FUNCTION_BLOCK EspPacketProcessor IMPLEMENTS ITF_Cyclic
VAR
	
	Udp							: ITF_UdpConnection;
	UdpReceiveBuffer			: REFERENCE TO ARRAY [0..TCPADS_MAXUDP_BUFFSIZE - 1] OF BYTE;
	LastCheckedIndex			: UDINT;
	List						: ITF_LinkedList;
	PacketsReceived				: ULINT;
	
	ReceivedPacketType			: BYTE;
	ReceivedPacketLocation		: PVOID;
	ReceivedPacketLength		: UINT;
	
	hr1							: HRESULT;
	OpenUdpConnection			: HRESULT;
	hr3							: HRESULT;
	
	TestPacket					: EspUdpPayload1;
	CurrentEsp32				: ITF_EspHost;
	
END_VAR
VAR CONSTANT
	StartDelimiter1				: BYTE := 2;
	StartDelimiter2				: BYTE := 181;
	EndDelimiter1				: BYTE := 91;
	EndDelimiter2				: BYTE := 03;
	PacketTypePosition			: BYTE := 37;
END_VAR

METHOD PRIVATE ClearBufferAtLocation : BOOL
VAR_INPUT
	PayloadLength			: UINT;
	PayloadLocation			: PVOID;
END_VAR
VAR
	i	: UDINT;
END_VAR

IF MEMSET(PayloadLocation, 0, PayloadLength) > 0 THEN

	ClearBufferAtLocation := TRUE;
	
ELSE
	
	ClearBufferAtLocation := FALSE;
	
END_IF

RETURN;
END_METHOD

METHOD ClearEntireBuffer : BOOL
VAR_INPUT
END_VAR
VAR
	i	: UDINT;
END_VAR

FOR i := 0 TO TCPADS_MAXUDP_BUFFSIZE - 1 BY 1 DO

	UdpReceiveBuffer[i] := 0;

END_FOR
END_METHOD

METHOD PRIVATE CopyPacketIntoStructure : BOOL
VAR_INPUT
	PayloadType				: BYTE;
	PayloadLength			: UINT;
	PayloadLocation			: PVOID;
END_VAR
CASE PayloadType OF
	
	1:
	
		MEMCPY(ADR(TestPacket), PayloadLocation, PayloadLength); 
		
		TestPacket.Start := HeaderEndianSwap(TestPacket.Start);
		
		TestPacket.End := TailEndianSwap(TestPacket.End);
		
		CopyPacketIntoStructure := TRUE;
		
		
		
	2:
	
		//
	
	
	
	3:
		
		//
	
	
	
END_CASE
END_METHOD

METHOD CreateEsp : BOOL
VAR_INPUT
END_VAR
END_METHOD

METHOD CyclicUpdate : BOOL
VAR
END_VAR

Udp.CyclicUpdate();
	

IF TryOpenConnection() = S_OK AND_THEN
	TryFindPacketInBuffer(ReceivedPacketType, ReceivedPacketLength, ReceivedPacketLocation) = S_OK AND_THEN
	CopyPacketIntoStructure(ReceivedPacketType, ReceivedPacketLength, ReceivedPacketLocation) AND_THEN 
	ClearBufferAtLocation(ReceivedPacketLength, ReceivedPacketLocation) THEN
	
	
	;
	
	
END_IF






// 
// hr1 := TryFindAPacketInBuffer(ReceivedPacketType, ReceivedPacketLength, ReceivedPacketLocation);
// 
// IF hr1 = S_OK THEN
// 	
// 	IF CopyPacketIntoStructure(ReceivedPacketType, ReceivedPacketLength, ReceivedPacketLocation) THEN
// 		
// 		ClearBufferAtLocation(ReceivedPacketLength, ReceivedPacketLocation);
// 		
// 	END_IF
// 
// END_IF
END_METHOD

//FB_Init is always available implicitly and it is used primarily for initialization.
//The return value is not evaluated. For a specific influence, you can also declare the
//methods explicitly and provide additional code there with the standard initialization
//code. You can evaluate the return value.
METHOD FB_Init: BOOL
VAR_INPUT
    bInitRetains: BOOL; // TRUE: the retain variables are initialized (reset warm / reset cold)
    bInCopyCode: BOOL;  // TRUE: the instance will be copied to the copy code afterward (online change)   
	UdpSocket	: ITF_UdpConnection;
	EspList		: ITF_LinkedList;
END_VAR
Udp := UdpSocket;
UdpReceiveBuffer REF= Udp.ReceiveBufferReference;
List := EspList;
END_METHOD

METHOD IsAcceptingData : BOOL
VAR_INPUT
END_VAR
IsAcceptingData := Udp.IsConnected();

RETURN;
END_METHOD

METHOD PRIVATE MatchUidToEsp : ITF_EspHost
VAR_INPUT
	Header	: EspUdpStart;
END_VAR
VAR
	Length	: UINT;
	i		: UINT;
	Node	: ITF_Node;
	Ptr		: POINTER TO EspHost;
	Esp		: ITF_EspHost;
	Uid		: ULINT;
END_VAR

Length := List.GetListLength();

IF Length = 0 THEN
	
	MatchUidToEsp := 0;
		
	RETURN;

END_IF

FOR i := 1 TO Length BY 1 DO

	Node := List.GetNode(i);	
	
	Ptr := Node.GetMyPointer();
	
	Esp := Ptr^;
	
	IF Esp = 0 THEN
		
		MatchUidToEsp := 0;
		
		RETURN;
		
	END_IF
	
	Uid := Esp.Uid;
	
	IF Uid = Header.SlaveUid THEN // = uid in buffer 
		
		MatchUidToEsp := Esp;
		
		RETURN;
		
	END_IF

END_FOR
END_METHOD

METHOD PRIVATE TryFindPacketInBuffer : HRESULT
VAR_INPUT
	PayloadType				: REFERENCE TO BYTE;
	PayloadLength			: REFERENCE TO UINT;
	PayloadLocation			: REFERENCE TO PVOID;
END_VAR
VAR
	i						: UDINT;
	Good					: BOOL;
END_VAR
TryFindPacketInBuffer := S_PENDING;

FOR i := LastCheckedIndex TO TCPADS_MAXUDP_BUFFSIZE - 1 BY 1 DO
	
	IF UdpReceiveBuffer[i] = StartDelimiter1 AND_THEN UdpReceiveBuffer[i + 1] = StartDelimiter2 THEN
		
		PayloadLength := BytesToUint(UdpReceiveBuffer[i + 2], UdpReceiveBuffer[i + 3]) + 50;
					
		PayloadType := UdpReceiveBuffer[i + PacketTypePosition];
		
		PayloadLocation := ADR(UdpReceiveBuffer[i]);
					
		IF PayloadLength = 0 OR PayloadType = 0 THEN
			
			TryFindPacketInBuffer := -1;
					
		ELSIF UdpReceiveBuffer[i + PayloadLength - 2] <> EndDelimiter1 OR UdpReceiveBuffer[i + PayloadLength - 1] <> EndDelimiter2 THEN
			
			TryFindPacketInBuffer := S_PENDING;
			
		ELSE
			
			PacketsReceived := PacketsReceived + 1;
			
			Good := TRUE;
			
		END_IF
		
		EXIT;
					
	END_IF

END_FOR

IF LastCheckedIndex > TCPADS_MAXUDP_BUFFSIZE - 1 THEN
	
	LastCheckedIndex := 0;
	
ELSE
	
	LastCheckedIndex := i;

END_IF

IF Good THEN
	
	TryFindPacketInBuffer := S_OK;
	
ELSE
	
	TryFindPacketInBuffer := S_PENDING;

END_IF

RETURN;
END_METHOD

METHOD PRIVATE TryOpenConnection : HRESULT
VAR_INPUT
END_VAR
TryOpenConnection := Udp.TryOpenConnection();

UdpReceiveBuffer REF= Udp.ReceiveBufferReference;

IF ADR(UdpReceiveBuffer) = 0 THEN

	TryOpenConnection := -1;	
	
END_IF

RETURN;
END_METHOD

END_FUNCTION_BLOCK

(* stored: Version 1.1.0.1
   POU EspPacketProcessor: Id {05be571e-be20-46fc-9aa3-6f0e1c571904}, SpecialFunc None
   Folder Private: Id {b3a90f2a-fb10-47d8-b27b-ed3a8f77b9e5}
   Folder Public: Id {a272a727-3988-4408-abfc-67103f70209e}
   Method ClearBufferAtLocation: Id {d451c427-ca4e-4e53-86c8-cf78b23bc920}
   Method ClearEntireBuffer: Id {5b97cea3-6cfc-44ef-848d-da951801b59a}
   Method CopyPacketIntoStructure: Id {a7cd640b-c057-4e56-87b7-444786445c11}
   Method CreateEsp: Id {0422dece-937d-4f2d-8f33-18aad4d44460}
   Method CyclicUpdate: Id {be97351d-5c68-4a8e-a83d-1e093e85b384}
   Method FB_Init: Id {de930b98-4376-4a46-92a0-2be25d257ea9}
   Method IsAcceptingData: Id {a8556bb5-22ae-4069-9b97-75360e7225b8}
   Method MatchUidToEsp: Id {a5acbb1d-0874-4cfb-aa5b-ecd39f0e29a6}
   Method TryFindPacketInBuffer: Id {b0962c32-b620-4d2c-8983-6c2de1d66f22}
   Method TryOpenConnection: Id {17cd8edb-53a2-4c77-9ed3-82863fdd1da4} *)
